// TIA Portal V19 export
FUNCTION_BLOCK "MotorS"   // FB124, LAD
TITLE = Fwd/Bkw Motor Managment FB
AUTHOR : TVA
FAMILY : Devices
NAME : Sys
VERSION : 4.2
// Motor FB with two directions.
// stored: Access Published, MemoryReserve 100, SetENOAutomatically false
   VAR_INPUT
      MotorCtrl : "Motor2Ctrl";
      ThermalProtectionA : Bool := FALSE;
      ThermalProtectionB : Bool := FALSE;
      FdbkRunning : Bool := FALSE;
      FeedbackTimeout : Time := T#500ms;
      ReversalTime : Time := T#500ms;
   END_VAR
   VAR_OUTPUT
      MotorSts : "MotorSts";
      BkwContactor : Bool;
      FwdContactor : Bool;
      Alarm : "MotorSAlr";
   END_VAR
   VAR
      InitDone : Bool;
      BkwDeny : Bool;
      FwdDeny : Bool;
      Ctrl_RunBkwContactor : Bool;
      Ctrl_RunFwdContactor : Bool;
      DelayContactorFeedbackON { S7_SetPoint := 'True'} : IEC_TIMER;
      DelayReversal { S7_SetPoint := 'True'} : IEC_TIMER;
   END_VAR
   VAR_TEMP
      AlarmPresence : Bool;
      RunPermitted : Bool;
   END_VAR
   VAR_TEMP   // added for the SCL form of the ladder/FBD networks
      _w1 : Bool;
   END_VAR
BEGIN

REGION Network 1: Alarm reset
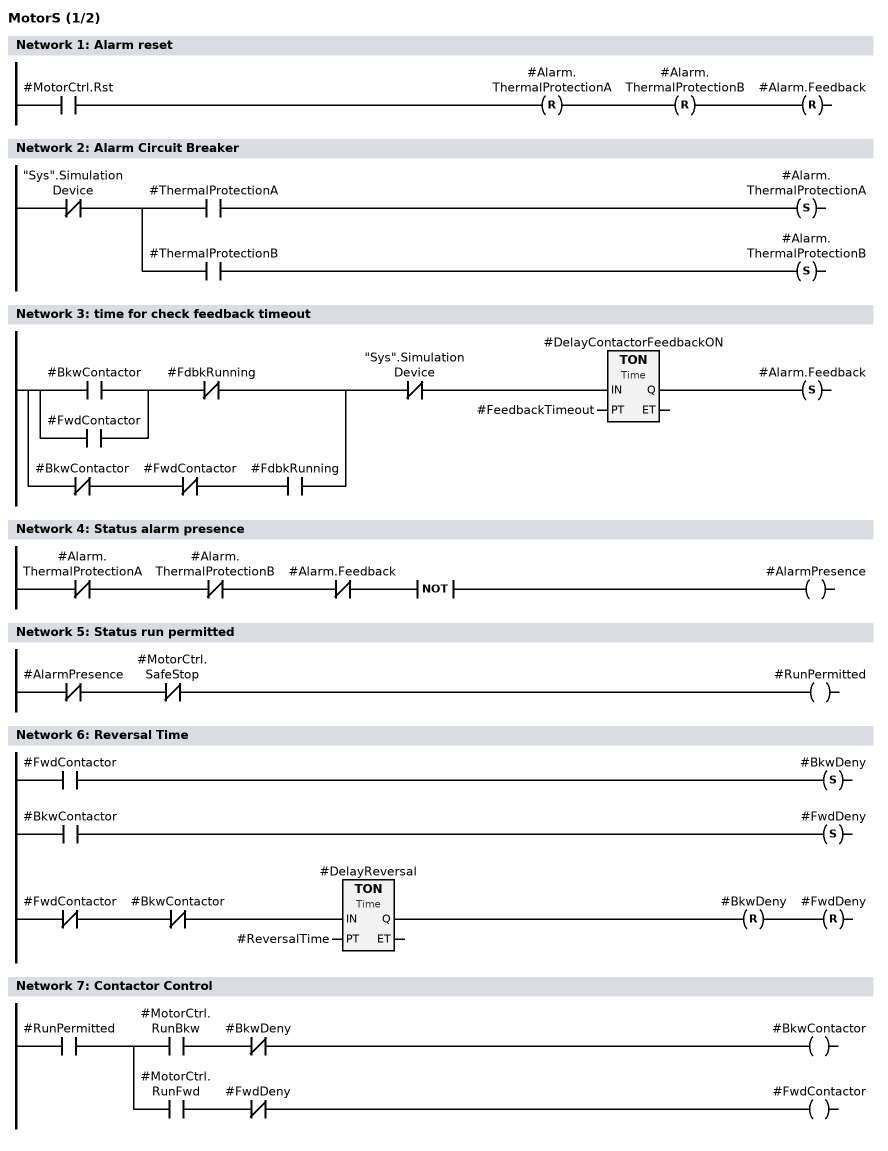
   RUNG wire#powerrail
      Contact( #MotorCtrl.Rst )
      R_Coil( #Alarm.ThermalProtectionA )
      R_Coil( #Alarm.ThermalProtectionB )
      R_Coil( #Alarm.Feedback )
   END_RUNG
   // the same network as SCL:
   IF #MotorCtrl.Rst THEN
       #Alarm.ThermalProtectionA := FALSE;
       #Alarm.ThermalProtectionB := FALSE;
       #Alarm.Feedback := FALSE;
   END_IF;
END_REGION

REGION Network 2: Alarm Circuit Breaker
   RUNG wire#powerrail
      I_Contact( "Sys".SimulationDevice )
      wire#w1
      Contact( #ThermalProtectionA )
      S_Coil( #Alarm.ThermalProtectionA )
   END_RUNG
   RUNG wire#w1
      Contact( #ThermalProtectionB )
      S_Coil( #Alarm.ThermalProtectionB )
   END_RUNG
   // the same network as SCL:
   #_w1 := NOT "Sys".SimulationDevice;
   IF #_w1 AND #ThermalProtectionA THEN #Alarm.ThermalProtectionA := TRUE; END_IF;
   IF #_w1 AND #ThermalProtectionB THEN #Alarm.ThermalProtectionB := TRUE; END_IF;
END_REGION

REGION Network 3: time for check feedback timeout
   RUNG wire#powerrail
      Contact( #BkwContactor )
      wire#w1
      I_Contact( #FdbkRunning )
      wire#w2
      I_Contact( "Sys".SimulationDevice )
      { S7_Templates := "time_type := Time" } #DelayContactorFeedbackON.TON(pt := #FeedbackTimeout, et =>)
      S_Coil( #Alarm.Feedback )
   END_RUNG
   RUNG wire#powerrail
      Contact( #FwdContactor )
   END_RUNG wire#w1
   RUNG wire#powerrail
      I_Contact( #BkwContactor )
      I_Contact( #FwdContactor )
      Contact( #FdbkRunning )
   END_RUNG wire#w2
   // the same network as SCL:
   #DelayContactorFeedbackON.TON(IN := (((#BkwContactor OR #FwdContactor) AND NOT #FdbkRunning) OR (NOT #BkwContactor AND NOT #FwdContactor AND #FdbkRunning)) AND NOT "Sys".SimulationDevice,
                           PT := #FeedbackTimeout);
   IF #DelayContactorFeedbackON.Q THEN #Alarm.Feedback := TRUE; END_IF;
END_REGION

REGION Network 4: Status alarm presence
   RUNG wire#powerrail
      I_Contact( #Alarm.ThermalProtectionA )
      I_Contact( #Alarm.ThermalProtectionB )
      I_Contact( #Alarm.Feedback )
      Not()
      Coil( #AlarmPresence )
   END_RUNG
   // the same network as SCL:
   #AlarmPresence := NOT (NOT #Alarm.ThermalProtectionA AND NOT #Alarm.ThermalProtectionB AND NOT #Alarm.Feedback);
END_REGION

REGION Network 5: Status run permitted
   RUNG wire#powerrail
      I_Contact( #AlarmPresence )
      I_Contact( #MotorCtrl.SafeStop )
      Coil( #RunPermitted )
   END_RUNG
   // the same network as SCL:
   #RunPermitted := NOT #AlarmPresence AND NOT #MotorCtrl.SafeStop;
END_REGION

REGION Network 6: Reversal Time
   RUNG wire#powerrail
      Contact( #FwdContactor )
      S_Coil( #BkwDeny )
   END_RUNG
   RUNG wire#powerrail
      Contact( #BkwContactor )
      S_Coil( #FwdDeny )
   END_RUNG
   RUNG wire#powerrail
      I_Contact( #FwdContactor )
      I_Contact( #BkwContactor )
      { S7_Templates := "time_type := Time" } #DelayReversal.TON(pt := #ReversalTime, et =>)
      R_Coil( #BkwDeny )
      R_Coil( #FwdDeny )
   END_RUNG
   // the same network as SCL:
   IF #FwdContactor THEN #BkwDeny := TRUE; END_IF;
   IF #BkwContactor THEN #FwdDeny := TRUE; END_IF;
   #DelayReversal.TON(IN := NOT #FwdContactor AND NOT #BkwContactor, PT := #ReversalTime);
   IF #DelayReversal.Q THEN
       #BkwDeny := FALSE;
       #FwdDeny := FALSE;
   END_IF;
END_REGION

REGION Network 7: Contactor Control
   RUNG wire#powerrail
      Contact( #RunPermitted )
      wire#w1
      Contact( #MotorCtrl.RunBkw )
      I_Contact( #BkwDeny )
      Coil( #BkwContactor )
   END_RUNG
   RUNG wire#w1
      Contact( #MotorCtrl.RunFwd )
      I_Contact( #FwdDeny )
      Coil( #FwdContactor )
   END_RUNG
   // the same network as SCL:
   #BkwContactor := #RunPermitted AND #MotorCtrl.RunBkw AND NOT #BkwDeny;
   #FwdContactor := #RunPermitted AND #MotorCtrl.RunFwd AND NOT #FwdDeny;
END_REGION

REGION Network 8: Coordination out
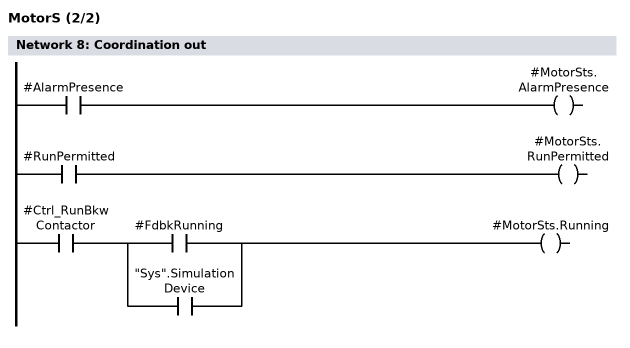
   RUNG wire#powerrail
      Contact( #AlarmPresence )
      Coil( #MotorSts.AlarmPresence )
   END_RUNG
   RUNG wire#powerrail
      Contact( #RunPermitted )
      Coil( #MotorSts.RunPermitted )
   END_RUNG
   RUNG wire#powerrail
      Contact( #Ctrl_RunBkwContactor )
      wire#w1
      Contact( #FdbkRunning )
      wire#w2
      Coil( #MotorSts.Running )
   END_RUNG
   RUNG wire#w1
      Contact( "Sys".SimulationDevice )
   END_RUNG wire#w2
   // the same network as SCL:
   #MotorSts.AlarmPresence := #AlarmPresence;
   #MotorSts.RunPermitted := #RunPermitted;
   #MotorSts.Running := #Ctrl_RunBkwContactor AND (#FdbkRunning OR "Sys".SimulationDevice);
END_REGION
END_FUNCTION_BLOCK
